# EPICS substitutions: iocs/MC05/MCApp/Db/SAI_EncoderLoss.substitutions
file /opt/epics/modules/SAI/db/SAI_EncoderLoss.template {
pattern {	P,		R,	AXIS,	SCAN, 		ASYNPORT, 	VARSTS, VARCLR}
        { 	"XF:06BMA-OP",		"{Mir:M3-Ax:",	"YU}Mtr","1 second",	"pmac",		"M181",	"M901"}
        { 	"XF:06BMA-OP",		"{Mir:M3-Ax:",	"YDO}Mtr","1 second",	"pmac",		"M281",	"M901"}
        { 	"XF:06BMA-OP",		"{Mir:M3-Ax:",	"YDI}Mtr","1 second",	"pmac",		"M381",	"M901"}
        { 	"XF:06BMA-OP",		"{Mir:M3-Ax:",	"XU}Mtr","1 second",	"pmac",		"M481",	"M901"}
        { 	"XF:06BMA-OP",		"{Mir:M3-Ax:",	"XD}Mtr","1 second",	"pmac",		"M581",	"M901"}
        { 	"XF:06BMA-BI",		"{Fltr:01-Ax:",	"Y1}Mtr","1 second",	"pmac",		"M681",	"M901"}
        { 	"XF:06BMA-BI",		"{Fltr:01-Ax:",	"Y2}Mtr","1 second",	"pmac",		"M781",	"M901"}
#        { 	"XF:06BMA-OP",		"{Mir:M3-Ax:",	"ZZZ}Mtr","1 second",	"pmac",		"M881",	"M901"}
}

#EOF
